PROGRAM PRG_Test
VAR
	McPower : MC_Power;
	McHalt : MC_Halt;
	
	Axis : AXIS_REF;
	
	nCurrentState : DINT := 0;
	
	bPower : BOOL := FALSE;
	bHalt : BOOL := FALSE;
END_VAR

McPower(
	Axis:= Axis, 
	Enable:= bPower, 
	Enable_Positive:= TRUE, 
	Enable_Negative:= TRUE, 
	Override:= 100, 
	BufferMode:= , 
	Options:= , 
	Status=> , 
	Busy=> , 
	Error=> , 
	ErrorID=> );
	
McHalt(
	Axis:= Axis, 
	Execute:= bHalt, 
	Deceleration:= , 
	Jerk:= , 
	BufferMode:= , 
	Options:= , 
	Done=> , 
	Busy=> , 
	Active=> , 
	CommandAborted=> , 
	Error=> , 
	ErrorID=> );

END_PROGRAM

(* stored: Version 1.1.0.1, ProductVersion 3.1.4024.15
   POU PRG_Test: Id {f6d34a71-0e55-4ba8-96ec-30398bce0da5}, SpecialFunc None *)
